PROGRAM S15_NG
VAR
	//工站
	station					: REFERENCE TO FB_Station:=fbstation[13];
	//气缸
	fbHOZCyl_1			:REFERENCE TO FB_Cylinder:=fbCylinder[27];	//	分料气缸1
	fbHOZCyl_2			:REFERENCE TO FB_Cylinder:=fbCylinder[28];	//	分料气缸2
	
	
	//延时
	arTonDelay :ARRAY[1..20] OF TON;
	//返回值
	UdiReturnValue :ARRAY[1..20] OF UDINT;
	
	
	
	i: INT;
	
	
END_VAR

A_Input();
Alarm();
Delay();
FlowAuto();
FlowInit();
General();
ILC();
TipAuto();
TipManual();
Z_Output();

ACTION A_Input:
//气缸
END_ACTION

ACTION Alarm:
//
station.adwAlarm[1].00:=station.xInitTimeout;	  			//S08Label 初始化超时
END_ACTION

ACTION Delay:
(*arTonDelay[01](IN:= , PT:=T#0.1S , Q=> , ET=> );*)//TipAuto使用
arTonDelay[02](IN:=  , PT:=T#1S , Q=> , ET=> );
arTonDelay[03](IN:=   , PT:=T#1S , Q=> , ET=> );
arTonDelay[04](IN:= , PT:=T#0.1S , Q=> , ET=> );
arTonDelay[05](IN:= , PT:=T#0.1S , Q=> , ET=> );
arTonDelay[06](IN:= , PT:=T#0.1S , Q=> , ET=> );
arTonDelay[07](IN:= , PT:=T#0.1S , Q=> , ET=> );
arTonDelay[08](IN:= , PT:=T#0.1S , Q=> , ET=> );
arTonDelay[09](IN:= , PT:=T#0.1S , Q=> , ET=> );
END_ACTION

ACTION FlowAuto:

//-----------------------------------------初始化是否完成判断----------------------------------------------
IF NOT station.xInitDone 
THEN
 	station.iStepAuto:=0;
 	station.xDone:=FALSE;
	station.xRunningOffProhibit := FALSE ;//运行中信号Off禁止
ELSIF station.xRunning  OR   station.xRunningOffProhibit
THEN
//-----------------------------------------动作步骤--------------------------------------------------------
CASE station.iStepAuto OF	  
	0: //----Home Step，等待启动----
		IF station.xDisabled 
			AND station.xCanRun 
			AND NOT fbMachine[1].xStopped 
			AND NOT station.xSingleRunning 
		THEN
			station.xDone:=TRUE;
		END_IF
		
		IF  station.xSingleRunning 
			OR station.xCanRun 
			AND NOT station.xDone 
			AND NOT station.xDisabled 
			AND NOT fbMachine[1].xStopped
		THEN
			station.xCycleEnable:=TRUE;
			station.xDone:= FALSE;  
			station.xRunningOffProhibit := TRUE ;//运行中信号Off禁止
			station.iStepAuto:= 10;
		END_IF
    10: //复位数据 
			station.iStepAuto:=20;
	
			
	
	999://----Single Run Finish----
			
		station.iStepAuto :=0;
		IF NOT station.xSingleContinuousRun THEN
			station.xSingleRunFlag:=FALSE;
		END_IF
		
		station.xCycleEnable:=FALSE;	
		station.xDone:=TRUE;
		station.xRunningOffProhibit := FALSE ;//运行中信号Off禁止
	ELSE
		;	
END_CASE



END_IF
END_ACTION

ACTION FlowInit:
IF NOT station.xIniting THEN
  station.iStepInit:=0;    
ELSE
//--------------------------------------------初始化步序----------------------------------
CASE station.iStepInit OF	
 0://  
  	IF station.xIniting THEN	
  	  station.iStepInit:=10;	
  	END_IF	
10://复位数据

100://	
    station.iStepInit:=999;	
999://初始化完成	
	station.iStepInit:=0;
	station.xInitDone:=TRUE;  
END_CASE
END_IF
END_ACTION

ACTION General:

END_ACTION

ACTION ILC:

//---------------------------------------------------工站可执行-------------------------------------------------------
station.xCanRun :=TRUE ;

//---------------------------------------------------气缸动作条件-------------------------------------------


//---------------------------------------------------伺服动作条件-------------------------------------------
END_ACTION

ACTION TipAuto:

//------------------------------------------------AutoTip Cylinder--------------------------------

//------------------------------------------------AutoTip Servo--------------------------------
//**************************************
END_ACTION

ACTION TipManual:
//--------------------------------------------ManualTip------------------------------------------------------

//-------------------------------------------气缸提示---------------------------------------------------------




/////////////////////////////////////////////////////////////////////////////////////////////////////////////////
END_ACTION

ACTION Z_Output:
(**************************气缸输出********************************)
END_ACTION

END_PROGRAM

(* stored: Version 1.1.0.1, ProductVersion 3.1.4024.9
   POU S15_NG: Id {fa03007f-9ac1-4b49-8987-777c7baa4a8b}, SpecialFunc None
   Action A_Input: Id {03aa5434-4f82-4612-9525-5439c5ebc821}
   Action Alarm: Id {c93c5b6a-db29-4dde-abc2-9023ce755d74}
   Action Delay: Id {2a42c8ab-5252-4e60-8c43-a3176ed90e84}
   Action FlowAuto: Id {13c9515b-61f3-4293-b7ba-ed91fbd853be}
   Action FlowInit: Id {bde57046-0c6b-4088-9111-b890c54bcabe}
   Action General: Id {18ca33ab-4a41-40cc-a10c-85884003a4c5}
   Action ILC: Id {76534184-9c70-4adc-9fee-3f36c06c66e3}
   Action TipAuto: Id {f79c7a30-b885-4edd-9ed5-9b2d935a7409}
   Action TipManual: Id {4b06f46d-7df0-47b3-9e69-6087ddee0dd5}
   Action Z_Output: Id {110fb2aa-1edf-4d7b-ba77-793b2ec8f7a5} *)
